// TIA Portal project "Pumpensicherung_ST" (V16)

(* hardware
DEVICE "S71500/ET200MP station_1"  S7-1500 station
   slot 0: "Rail_0"  Rack  6ES7 590-1***0-0AA0
   slot 1: "PLC_1"  CPU 1511-1 PN  6ES7 511-1AK00-0AB0  V1.8
      slot 3: "CPU display_1"  6ES7591-1AA00-0AA0
      slot 32768: "PROFINET interface_1"  X1
         slot 32769: "Port_1"  X1 P1
         slot 32770: "Port_2"  X1 P2
   slot 2: "DI 16x24VDC BA_1"  DI 16x24VDC BA  6ES7 521-1BH10-0AA0  V1.1
   slot 3: "DQ 8x24VDC/2A HF_1"  DQ 8x24VDC/2A HF  6ES7 522-1BF00-0AB0  V2.2
   slot 4: "AI 4xU/I/RTD/TC ST_1"  AI 4xU/I/RTD/TC ST  6ES7 531-7QD00-0AB0  V1.0
*)

// ===== PLC "PLC_1"  CPU 1511-1 PN =====

VAR_GLOBAL   // PLC tag table "Default tag table"
   "Strömungsschalter" AT %I0.0 : Bool;
   "Alarm-Reset" AT %I0.1 : Bool;
   "Alarmstummschalter" AT %I0.2 : Bool;
   "Hand-taste" AT %I0.3 : Bool;
   "Aus-Taste" AT %I0.4 : Bool;
   "Auto-Taste" AT %I0.5 : Bool;
   "Pumpe" AT %Q0.0 : Bool;
   "Strömungsschalterdefektleuchte" AT %Q0.1 : Bool;
   "Drucksensordefektleuchte" AT %Q0.2 : Bool;
   "Strömungschalter_Bit" AT %M4.0 : Bool;
   "Alarm-Reset_Bit" AT %M4.1 : Bool;
   "Alarmstummschalter_Bit" AT %M4.2 : Bool;
   "Hand_Taste_Bit" AT %M4.3 : Bool;
   "Aus_Taste_Bit" AT %M4.4 : Bool;
   "Auto_Taste_Bit" AT %M4.5 : Bool;
   "HOA_Modi" AT %MW6 : Int;   // 0 = AUS ; 1 = HAND ; 2 = AUTO
   "ONS1" AT %M4.6 : Bool;
   "ONS2" AT %M4.7 : Bool;
   "ONS3" AT %M5.0 : Bool;
   "Modus_vor_Hand" AT %MW8 : Int;
   "ONS4" AT %M5.3 : Bool;
   "Pumpe_AUTO_MODUS" AT %MW10 : Int;   // 1 = AN ; 0 = AUS
   "Pumpe_Interrupt" AT %M5.4 : Bool;
   "Strömungsschalterdefektleuchte_Bit" AT %M5.5 : Bool;
   "Pumpe_Bit" AT %M5.6 : Bool;
   "Drucksensordefektleuchte_Bit" AT %M5.7 : Bool;
   "Strömungsstörung_Alarmmeldung_Bit" AT %M12.0 : Bool;
   "Überdrucklalarmmeldung_Bit" AT %M12.1 : Bool;
   "Drucksensor_Ersatz" AT %MW14 : Int;
   "Druck in PSI" AT %MD16 : Real;
   "Alarm_Bit" AT %M0.0 : Bool;
   "One Shot" AT %M0.1 : Bool;
END_VAR

DATA_BLOCK "IO_DB"   // DB1
{ S7_Optimized_Access := 'TRUE' }
VERSION : 0.1
// stored: InstanceOfName IO
"IO"
BEGIN
END_DATA_BLOCK

DATA_BLOCK "HOA_DB"   // DB2
{ S7_Optimized_Access := 'TRUE' }
VERSION : 0.1
// stored: InstanceOfName HOA
"HOA"
BEGIN
END_DATA_BLOCK

DATA_BLOCK "Steuerung_DB"   // DB4
{ S7_Optimized_Access := 'TRUE' }
VERSION : 0.1
// stored: InstanceOfName Steuerung
"Steuerung"
BEGIN
END_DATA_BLOCK

DATA_BLOCK "Alarms_DB"   // DB13
{ S7_Optimized_Access := 'TRUE' }
VERSION : 0.1
// stored: InstanceOfName Alarms
"Alarms"
BEGIN
END_DATA_BLOCK

// folder: System blocks/Program resources

DATA_BLOCK "Pumpe_Aus_Verzögerung"   // DB3
{ S7_Optimized_Access := 'TRUE' }
AUTHOR : Simatic
FAMILY : IEC
NAME : IEC_TMR
VERSION : 1.0
// stored: InstanceOfName IEC_TIMER
"IEC_TIMER"
BEGIN
END_DATA_BLOCK

DATA_BLOCK "Pumpe_An_Verzögerung"   // DB5
{ S7_Optimized_Access := 'TRUE' }
AUTHOR : Simatic
FAMILY : IEC
NAME : IEC_TMR
VERSION : 1.0
// stored: InstanceOfName IEC_TIMER
"IEC_TIMER"
BEGIN
END_DATA_BLOCK

DATA_BLOCK "Überdruckalarm"   // DB10
{ S7_Optimized_Access := 'TRUE' }
AUTHOR : Simatic
FAMILY : IEC
NAME : IEC_TMR
VERSION : 1.0
// stored: InstanceOfName IEC_TIMER
"IEC_TIMER"
BEGIN
END_DATA_BLOCK

DATA_BLOCK "Strömungsstörungalarm"   // DB15
{ S7_Optimized_Access := 'TRUE' }
AUTHOR : Simatic
FAMILY : IEC
NAME : IEC_TMR
VERSION : 1.0
// stored: InstanceOfName IEC_TIMER
"IEC_TIMER"
BEGIN
END_DATA_BLOCK

// folder: (top level)

FUNCTION_BLOCK "IO"   // FB1, SCL
{ S7_Optimized_Access := 'TRUE' }
VERSION : 0.1
   VAR
      Normalisierter_Wert : Real;
   END_VAR
BEGIN
   // Eingänge
   IF "Strömungsschalter" THEN
       "Strömungschalter_Bit" := TRUE;
   ELSE
       "Strömungschalter_Bit" := FALSE;
   END_IF;

   IF "Alarm-Reset" THEN
       "Alarm-Reset_Bit" := TRUE;
   ELSE
       "Alarm-Reset_Bit" := FALSE;
   END_IF;

   IF "Alarmstummschalter" THEN
       "Alarmstummschalter_Bit" := TRUE;
   ELSE
       "Alarmstummschalter_Bit" := FALSE;
   END_IF;

   IF "Hand-taste" THEN
       "Hand_Taste_Bit" := TRUE;
   ELSE
       "Hand_Taste_Bit" := FALSE;
   END_IF;

   IF "Aus-Taste" THEN
       "Aus_Taste_Bit" := TRUE;
   ELSE
       "Aus_Taste_Bit" := FALSE;
   END_IF;

   IF "Auto-Taste" THEN
       "Auto_Taste_Bit" := TRUE;
   ELSE
       "Auto_Taste_Bit" := FALSE;
   END_IF;

   #Normalisierter_Wert := NORM_X(MIN := 0, VALUE := "Drucksensor_Ersatz", MAX := 27648);
   "Druck in PSI" := SCALE_X(MIN := 0.0, VALUE := #Normalisierter_Wert, MAX := 55.0);

   // Ausgänge
   IF "Pumpe_Bit" THEN
       "Pumpe" := TRUE;
   ELSE
       "Pumpe" := FALSE;
   END_IF;

   IF "Strömungsschalterdefektleuchte_Bit" THEN
       "Strömungsschalterdefektleuchte" := TRUE;
   ELSE
       "Strömungsschalterdefektleuchte" := FALSE;
   END_IF;

   IF "Drucksensordefektleuchte_Bit" THEN
       "Drucksensordefektleuchte" := TRUE;
   ELSE
       "Drucksensordefektleuchte" := FALSE;
   END_IF;
END_FUNCTION_BLOCK

FUNCTION_BLOCK "HOA"   // FB2, SCL
{ S7_Optimized_Access := 'TRUE' }
VERSION : 0.1
   VAR
      AUTO_ONS_FLAG_1 : Bool;
      AUTO_ONS_FLAG_2 : Bool;
      AUS_ONS_FLAG_1 : Bool;
      HAND_ONS_FLAG_1 : Bool;
      HAND_ONS_FLAG_2 : Bool;
   END_VAR
BEGIN
   // HOA AUTO
   IF "Auto_Taste_Bit" AND NOT "Alarm_Bit" AND NOT #AUTO_ONS_FLAG_1 THEN
       "HOA_Modi" := 2;
       #AUTO_ONS_FLAG_1:= TRUE;

   END_IF;
   IF NOT "Auto_Taste_Bit" AND NOT "Alarm_Bit" THEN
       #AUTO_ONS_FLAG_1:= FALSE;
   END_IF;

   IF "HOA_Modi" = 2 AND NOT #AUTO_ONS_FLAG_2  THEN
       "Pumpe_AUTO_MODUS" := 1;
       #AUTO_ONS_FLAG_2 := TRUE;
   END_IF;
   IF "HOA_Modi" <> 2 THEN
       #AUTO_ONS_FLAG_2 := FALSE;
   END_IF;

   // HOA AUS
   IF "Aus_Taste_Bit" AND NOT #AUS_ONS_FLAG_1 THEN
       "HOA_Modi" := 0;
       "Modus_vor_Hand" := "HOA_Modi";
       "Pumpe_AUTO_MODUS" := "HOA_Modi";
       #AUS_ONS_FLAG_1 := TRUE;
   END_IF;
   IF NOT "Aus_Taste_Bit" THEN
       #AUS_ONS_FLAG_1 := FALSE;
   END_IF;


   // HOA HAND
   IF "Hand_Taste_Bit" AND NOT "Alarm_Bit" AND NOT #HAND_ONS_FLAG_1 THEN
       "Modus_vor_Hand" := "HOA_Modi";
       "HOA_Modi" := 1;
       #HAND_ONS_FLAG_1 := TRUE;
   END_IF;
   IF NOT "Hand_Taste_Bit" AND NOT "Alarm_Bit" THEN
       #HAND_ONS_FLAG_1 := FALSE;
   END_IF;

   IF "HOA_Modi" = 1 AND NOT "Hand_Taste_Bit" AND NOT #HAND_ONS_FLAG_2 THEN
       "HOA_Modi" := "Modus_vor_Hand";
       #HAND_ONS_FLAG_2 := TRUE;
   END_IF;
   IF "HOA_Modi" <> 1 AND NOT "Hand_Taste_Bit" THEN
       #HAND_ONS_FLAG_2 := FALSE;
   END_IF;
END_FUNCTION_BLOCK

FUNCTION_BLOCK "Steuerung"   // FB3, SCL
{ S7_Optimized_Access := 'TRUE' }
VERSION : 0.1
   VAR
      AUTO_STEUERUNG_ONS_FLAG_1 : Bool;
      Pumpe_Auto_Trigger : Bool;
      TON_OUTPUT : Bool;
      Pumpe_AUTO_BIT : Bool;
      TON2_OUTPUT : Bool;
      Pumpe_HAND_BIT : Bool;
      Pumpe_Aus_Verzögerung_TON : Bool;
      Pumpe_An_Verzögerung_TON : Bool;
      AUTO_Trigger_Condition : Bool;
      HAND_Trigger_Condition : Bool;
      Pumpe_Hand_Trigger : Bool;
      ONS_Strömung : Bool;
      ONS_Reset_Q : Bool;
      ONS_Strömung_Q : Bool;
      ONS_Druck_Q : Bool;
   END_VAR
BEGIN
   // Auto Steuerung
   #AUTO_Trigger_Condition := ("HOA_Modi" = 2) AND ("Pumpe_AUTO_MODUS" = 1) AND NOT "Alarm_Bit";
   "Pumpe_Trigger"(CLK:=#AUTO_Trigger_Condition,
                   Q=>#Pumpe_Auto_Trigger);

   IF "HOA_Modi" = 2 AND "Pumpe_AUTO_MODUS" = 1 AND NOT "Alarm_Bit" THEN
       #Pumpe_Aus_Verzögerung_TON := TRUE;
   ELSE
       #Pumpe_Aus_Verzögerung_TON := FALSE;
   END_IF;

       "Pumpe_Aus_Verzögerung".TON(IN := #Pumpe_Aus_Verzögerung_TON,
                                   PT := T#30s,
                                   Q => #TON_OUTPUT);

       IF #TON_OUTPUT THEN
           "Pumpe_Interrupt" := TRUE;
           "Pumpe_AUTO_MODUS" := 0;
       END_IF;


   IF #Pumpe_Auto_Trigger OR ("Pumpe_Bit" AND "HOA_Modi" = 2 AND NOT "Alarm_Bit" AND NOT "Pumpe_Interrupt") THEN
       #Pumpe_AUTO_BIT := TRUE;
   ELSE
       #Pumpe_AUTO_BIT := FALSE;
   END_IF;

   IF "HOA_Modi" = 2 AND "Pumpe_AUTO_MODUS" = 0 AND NOT "Alarm_Bit" THEN
       #Pumpe_An_Verzögerung_TON := TRUE;
   ELSE
       #Pumpe_An_Verzögerung_TON := FALSE;
   END_IF;
       "Pumpe_An_Verzögerung".TON(IN := #Pumpe_An_Verzögerung_TON,
                                  PT:=T#10s,
                                  Q=>#TON2_OUTPUT);
       IF #TON2_OUTPUT THEN
           "Pumpe_AUTO_MODUS" := 1;
           "Pumpe_Interrupt" := False;
       END_IF;

   //HAND Steuerung
       #HAND_Trigger_Condition := ("HOA_Modi" = 1) AND NOT "Alarm_Bit";
   "HAND_Pumpe_Trigger"(CLK:=#HAND_Trigger_Condition,
                        Q=>#Pumpe_Hand_Trigger);

   IF #Pumpe_Hand_Trigger OR ("Pumpe_Bit" AND NOT "Alarm_Bit" AND "HOA_Modi" = 1) THEN
       #Pumpe_HAND_BIT := TRUE;
   ELSE
       #Pumpe_HAND_BIT := FALSE;
   END_IF;


   // Pumpensteuerung
   IF "HOA_Modi" <> 0 AND (#Pumpe_AUTO_BIT OR #Pumpe_HAND_BIT) THEN
       "Pumpe_Bit" := TRUE;
   ELSE
       "Pumpe_Bit" := False;
   END_IF;
   // Alarmbeleuchtung
   "ONS_Strömung"(CLK := "Strömungsstörung_Alarmmeldung_Bit",
                  Q => #ONS_Strömung_Q);
   IF ("Strömungsschalterdefektleuchte_Bit" AND NOT "Alarmstummschalter_Bit") OR #ONS_Strömung_Q THEN
       "Strömungsschalterdefektleuchte_Bit" := TRUE;
   ELSE
       "Strömungsschalterdefektleuchte_Bit" := FALSE;
   END_IF;

   "ONS_Druck"(CLK:="Überdrucklalarmmeldung_Bit",
               Q=>#ONS_Druck_Q);
   IF ("Drucksensordefektleuchte_Bit" AND NOT "Alarmstummschalter_Bit") OR #ONS_Druck_Q THEN
       "Drucksensordefektleuchte_Bit" := TRUE;
   ELSE
       "Drucksensordefektleuchte_Bit" := FALSE;
   END_IF;

   // Alarmreset
   "ONS_Reset"(CLK:="Alarm-Reset_Bit",
               Q=>#ONS_Reset_Q);

   IF #ONS_Reset_Q THEN
       "HOA_Modi" := 0;
       "Modus_vor_Hand" := 0;
   END_IF;
END_FUNCTION_BLOCK

FUNCTION_BLOCK "Alarms"   // FB4, SCL
{ S7_Optimized_Access := 'TRUE' }
VERSION : 0.1
   VAR
      Überdruckalarm_IN : Bool;
      Überdruckalarm_Q : Bool;
      Überdruckalarm_Trigger_ONS : Bool;
      Überdruckalarmmeldung_Trigger : Bool;
      Überdruck_Alarm : Bool;
      Strömungsstörungalarm_IN : Bool;
      Strömungsstörungalarm_Q : Bool;
      Strömungsstörung_Alarm_Trigger : Bool;
      Strömungsstörung_Alarmmeldung_Trigger : Bool;
      Strömungsstörung_Alarm : Bool;
   END_VAR
BEGIN
   // DRUCK_ALARM
   IF "Druck in PSI" > 30.0  THEN
       #Überdruckalarm_IN := TRUE;
   ELSE
       #Überdruckalarm_IN := FALSE;

   END_IF;
   "Überdruckalarm".TON(IN:=#Überdruckalarm_IN,
                        PT:=T#5s,
                        Q=>#Überdruckalarm_Q);
   "Überdruckalarm_Trigger"(CLK:=#Überdruckalarm_Q,
                            Q=>#Überdruckalarm_Trigger_ONS);
   "Überdruckalarmmeldung_ONS"(CLK:=#Überdruckalarm_Q,
                               Q=>#Überdruckalarmmeldung_Trigger);

   IF (#Überdruckalarm_Trigger_ONS) OR (#Überdruck_Alarm AND NOT "Alarm-Reset_Bit") THEN
       #Überdruck_Alarm := TRUE;
   ELSE
       #Überdruck_Alarm := FALSE;
   END_IF;

   IF (#Überdruckalarmmeldung_Trigger) OR ("Überdrucklalarmmeldung_Bit" AND NOT "Alarm-Reset_Bit" AND NOT "Alarmstummschalter_Bit") THEN
       "Überdrucklalarmmeldung_Bit" := TRUE;
   ELSE
       "Überdrucklalarmmeldung_Bit" := FALSE;
   END_IF;

   // Strömungs_ALARM
   IF ("HOA_Modi" = 1 OR "HOA_Modi" = 2) AND NOT "Strömungschalter_Bit" THEN
       #Strömungsstörungalarm_IN := TRUE;
   ELSE
       #Strömungsstörungalarm_IN := FALSE;
   END_IF;
   "Strömungsstörungalarm".TON(IN:=#Strömungsstörungalarm_IN,
                               PT:=T#5s,
                               Q=>#Strömungsstörungalarm_Q);

   "Strömungsstörung_Alarm_Trigger_ONS"(CLK:=#Strömungsstörungalarm_Q,
                                        Q=>#Strömungsstörung_Alarm_Trigger);
   "Strömungsstörung_Alarmmeldung_Trigger_ONS"(CLK:=#Strömungsstörungalarm_Q,
                                               Q=>#Strömungsstörung_Alarmmeldung_Trigger);

   IF(#Strömungsstörung_Alarm_Trigger) OR (#Strömungsstörung_Alarm AND NOT "Alarm-Reset_Bit") THEN
       #Strömungsstörung_Alarm := TRUE;
   ELSE
       #Strömungsstörung_Alarm := FALSE;
   END_IF;

   IF (#Strömungsstörung_Alarmmeldung_Trigger)OR("Strömungsstörung_Alarmmeldung_Bit" AND NOT "Alarm-Reset_Bit" AND NOT "Alarmstummschalter_Bit") THEN
       "Strömungsstörung_Alarmmeldung_Bit" := TRUE;
   ELSE
       "Strömungsstörung_Alarmmeldung_Bit" := FALSE;
   END_IF;

   // ALARM_BIT
   IF (#Strömungsstörung_Alarm) OR (#Überdruck_Alarm) THEN
       "Alarm_Bit" := TRUE;
   ELSE
       "Alarm_Bit" := FALSE;
   END_IF;
END_FUNCTION_BLOCK

ORGANIZATION_BLOCK "Main"   // OB1, LAD, ProgramCycle
TITLE = "Main Program Sweep (Cycle)"
{ S7_Optimized_Access := 'TRUE' }
VERSION : 0.1
// PROJEKTBESCHREIBUNG: BEI DIESEM PROJEKT GEHT ES UM DIE SICHERHEIT DER PUMPE. DIE 
// SICHERHEIT DER PUMPE WIRD DURCH EINE KOMBINATION VON ZWEI SENSOREN GEWÄHRLEISTET:1) STRÖMUNGSSCHALTER 2) DRUCKSENSOR .DER STRÖMUNGSSCHALTER WIRD VOR DER PUMPE UND DER DRUCKSENSOR NACH DEM PUMPE MONTIERT. SOBALD DIE PUMPE AN IST UND FÜR FÜNF SEKUNDEN LÄUFT, WIRD ES FESTGESTELLT, OB DER STRÖMUNGSCHALTER GESCHLOSSEN IST UND/ODER OB DER DRUCK NACH DER PUMPE KLEINER ALS 30 PSI IST. WENN ES NICHT DER FALL IST, WIRD EIN ALARM AUSGELÖST UND DIE PUMPE AUSGESCHALTET. SOLANGE DANN DER ALARM-RESET NICHT BETÄTIGT WIRD, KANN DIE PUMPE NICHT WIEDER IM BETRIEB GENOMMEN WERDEN. AUßERDEM WIRD DIE PUMP MITTELS HAND/AUTOMATIK/AUS SCHALTER BETRIEBEN. SOLANGE DIE HANDTASTE GEDRUCKT BLEIBT, LÄUFT DIE PUMPE. SOBALD DIE HANDTASTE LOSGELASSEN WIRD GEHT DIE PUMPE WIRD IM MODUS, DAS VOR DEM HAND-MODUS AKTIV WAR. IN AUTO-MODUS LÄUFT DIE PUMPE IN EINEM ZYKLUS. DAS HEIßT, DIE PUMPE IST FÜR 30 SEKUNDEN AN UND DANN BLEIBT AUS FÜR 10 SEKUNDEN UND DANN WIEDER AN FÜR 30 SEKUNDEN UND SO WEITER. IM OFF-MODUS (AUS) BLEIBT DIE PUMPE AUS.
// 
// TESTKRITERIEN:
// 1) ZUNÄCHST BLEIBT DIE PUMPE AUS. SETZE DRUCKERSATZ AUF 13824 UND DER DRUCK SOLLTE 27,5 PSI BETRAGEN.
// 2) HANDTASTE WIRD GEDRUCKT BZW EINGESCHALTET. DIE PUMPE GEHT AN UND BLEIBT AN FÜR 5 SEKUNDEN UND DANN WIEDER AUS. DER ALARM WIRD AUSGELÖST UND DIE STRÖMUNGSSCHALTERDEFEKTLEUCHTE LEUCHTET.
// 3) HANDTASTE WIRD LOSGELASSEN UND DER ALARMSTUMMSCHALTER WIRD BETÄTIGT UND DIE LEUCHTE GEHT WIEDER AUS. HANDTASTE WIRD FÜR EINIGE SEKUNDEN GEDRUCKT UND WIEDER LOSGELASSEN ABER DIE PUMPE GEHT NICHT AN.
// 4) AUTOTASTE WIRD GETOGGELT. DIE PUMPEZYKLUS SOLLTE NICHT AN GEHEN
// 5) ALARMRESET WIRD BETÄTIGT UND DANN WIRD STRÖMUNGSCHALTER GESCHALTET. NUN WIRD AUTOTASTE GETOGGELT. DIE PUMPE SOLLTE IM ZYKLUS LAUFEN. 
// 6) NUN WIRD HANDTASTE GEDRUCKT FÜR UNGEFÄHR 20 SEKUNDEN. DIE PUMPE SOLLTE AUS DEM ZYKLUS RAUS UND STÄNDIG LAUFEN. WIRD DIE HANDTASTE WIEDER GELASSEN SOLLTE DIE PUMPE WIRD IM ZYKLUS LAUFEN.
// 7) SETZE DRUCKERSATZ AUF 16876 UND DIE PUMPE SOLLTE NACH 5 SEKUNDEN AUS GEHEN. DER ALARM WIRD AUSGELÖST UND DIE DRUCKSENSORDEFEKTLEUCHTE LEUCHTET. DER DRUCKWERT BETRÄGT 33,5 PSI.
   VAR_INPUT
      Initial_Call : Bool;   // Initial call of this OB
      Remanence : Bool;   // =True, if remanent data are available
   END_VAR
BEGIN

REGION Network 1
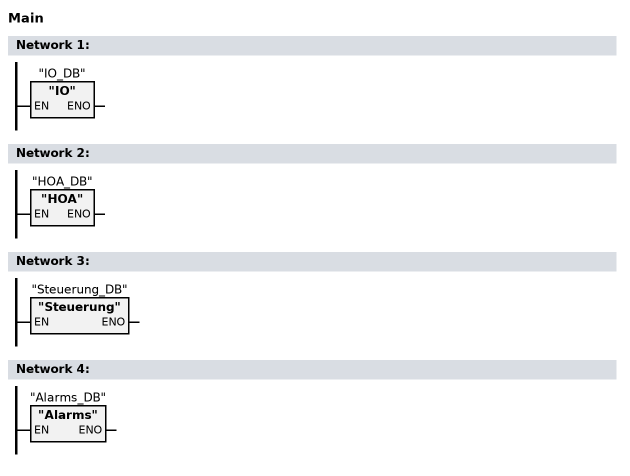
   RUNG wire#powerrail
      "IO_DB"()
   END_RUNG
   // the same network as SCL:
   "IO_DB"();   // "IO"
END_REGION

REGION Network 2
   RUNG wire#powerrail
      "HOA_DB"()
   END_RUNG
   // the same network as SCL:
   "HOA_DB"();   // "HOA"
END_REGION

REGION Network 3
   RUNG wire#powerrail
      "Steuerung_DB"()
   END_RUNG
   // the same network as SCL:
   "Steuerung_DB"();   // "Steuerung"
END_REGION

REGION Network 4
   RUNG wire#powerrail
      "Alarms_DB"()
   END_RUNG
   // the same network as SCL:
   "Alarms_DB"();   // "Alarms"
END_REGION
END_ORGANIZATION_BLOCK